FUNCTION_BLOCK FB_ElectricityMeter
VAR_INPUT
END_VAR
VAR_OUTPUT
END_VAR
VAR
END_VAR

END_FUNCTION_BLOCK

(* stored: Version 1.1.0.1, ProductVersion 3.1.4024.10
   POU FB_ElectricityMeter: Id {71edd3b2-6767-4a7d-bd1b-bd5eb886f3be}, SpecialFunc None *)
